TYPE "Positioning_MOL_Machine_DataIn"
VERSION : 0.1
// Block: Positioning_MOL_Machine_DataIn
   STRUCT
      PB : Ax_PB;
      LS_Minus : Bool;
      LS_Plus : Bool;
      M1_TherrmalProtection : Bool;
      M2_TherrmalProtection : Bool;
      M1M2_Feedback : Bool;
   END_STRUCT;

END_TYPE
